# B&R Automation Studio project acoposTrak_simple_control
Automation Studio 4.9.2.46; technology packages: mappMotion 5.12.2, mappView 5.12.1

## Configuration Config1

CPU X20CP3687X, AutomationRuntime C4.90, Build 4.1.2, Vc V4.72.2

### Task classes (Cpu.sw)
```
Cyclic#1 (cycle 2000 us, tolerance 0 us):
  tCTRL_m <- Technology.tCTRL_m.prg
DataObjects: McAcpSys
Binaries: FWRules, McAcpSim, arcoal, arsvcreg, TCData, McAcpDrv, McProfGen, arflatprv, udbdef, iomap, Config_1, arconfig, asfw, ashwac, sysconf, Role, ashwd, User, Config_3, Config_2
Libraries: McBase, McAxis, McAcpTrak, AsBrStr, runtime, astime, fileio, powerlnk, asieccon, standard, asstring
```

### Hardware
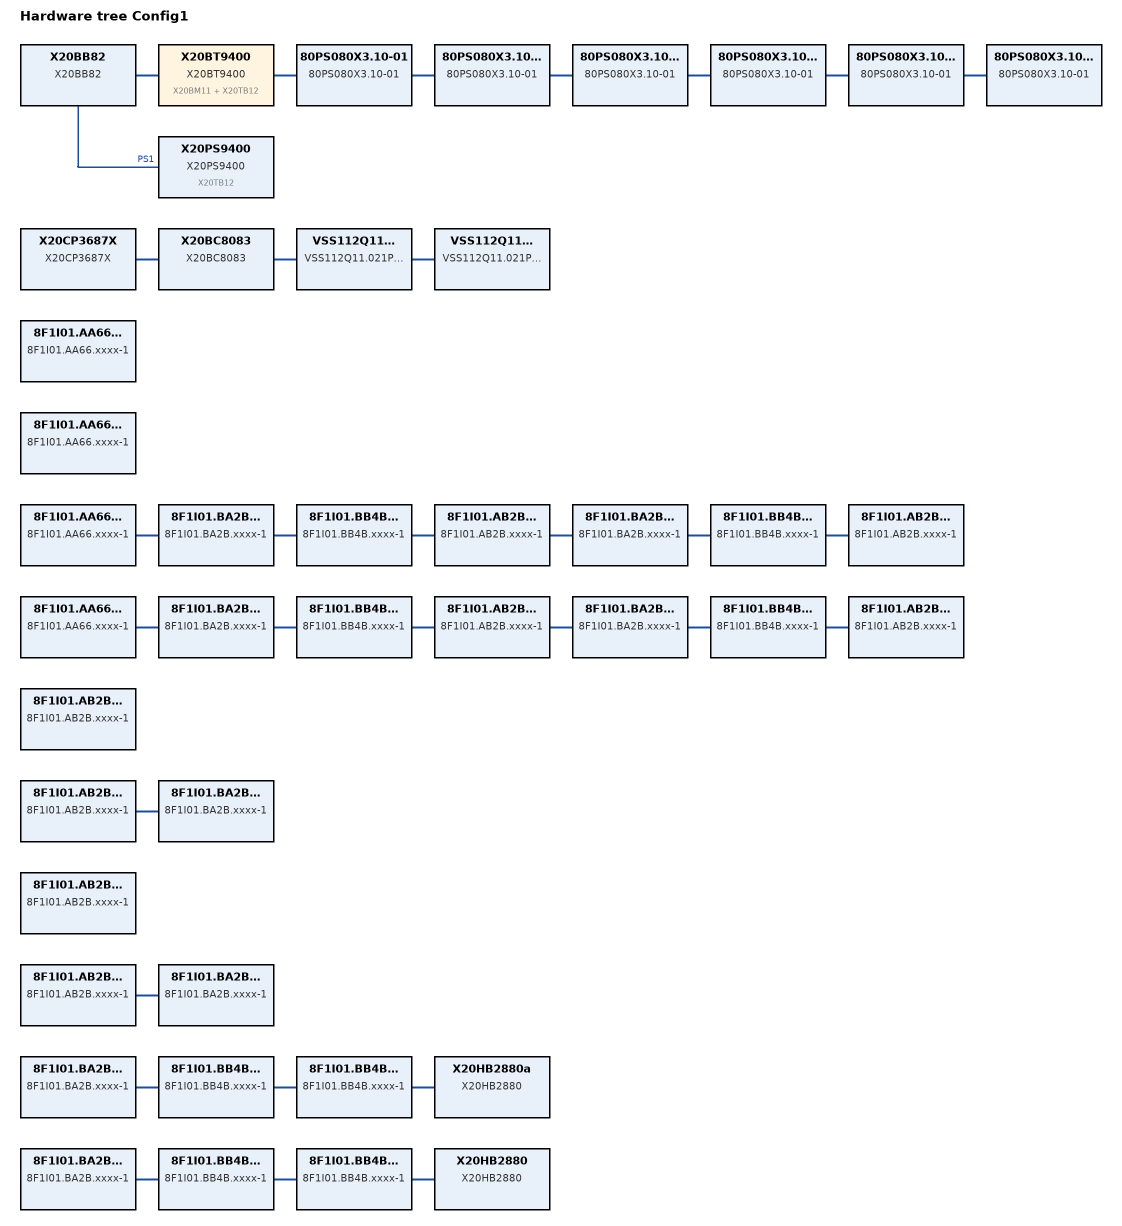
```
80PS080X3.10-01 : 80PS080X3.10-01 v1.3.0.0  [X2X1 -> X20BT9400.X2X1 [Cable Type=X2XCable, Length=10, Version=1.0.0.3]]
  Supervision = off
  VoltageSet01 = 60
80PS080X3.10-01a : 80PS080X3.10-01 v1.3.0.0  [X2X1 -> 80PS080X3.10-01.X2X2 [Cable Type=X2XCable, Length=10, Version=1.0.0.3]]
  ParallelMode01 = on
  VoltageSet01 = 60
80PS080X3.10-01b : 80PS080X3.10-01 v1.3.0.0  [X2X1 -> 80PS080X3.10-01a.X2X2 [Cable Type=X2XCable, Length=10, Version=1.0.0.3]]
  ParallelMode01 = on
  VoltageSet01 = 60
80PS080X3.10-01c : 80PS080X3.10-01 v1.3.0.0  [X2X1 -> 80PS080X3.10-01b.X2X2 [Cable Type=X2XCable, Length=10, Version=1.0.0.3]]
  ParallelMode01 = on
  VoltageSet01 = 60
80PS080X3.10-01d : 80PS080X3.10-01 v1.3.0.0  [X2X1 -> 80PS080X3.10-01c.X2X2 [Cable Type=X2XCable, Length=10, Version=1.0.0.3]]
  ParallelMode01 = on
  VoltageSet01 = 60
80PS080X3.10-01e : 80PS080X3.10-01 v1.3.0.0  [X2X1 -> 80PS080X3.10-01d.X2X2 [Cable Type=X2XCable, Length=10, Version=1.0.0.3]]
  ParallelMode01 = on
  VoltageSet01 = 60
8F1I01.AA66.xxxx-1 : 8F1I01.AA66.xxxx-1 v1.0.0.2  [PLK1 -> 8F1I01.AB2B.xxxx-1.PLK2 [Cable Type=PowerlinkCable, Length=10, Version=1.0.0.3]]
  DriveConfiguration:
    McTypeID = LLMConfig
  DriveConfiguration/Segment:
    Shape = STRAIGHT660
    SegmentReference = Seg_A_1
    StopReaction = UseAssemblySetting
    SpeedFilter = UseAssemblySetting
8F1I01.AA66.xxxx-1a : 8F1I01.AA66.xxxx-1 v1.0.0.2  [PLK1 -> 8F1I01.AB2B.xxxx-1b.PLK2 [Cable Type=PowerlinkCable, Length=10, Version=1.0.0.3]]
  DriveConfiguration:
    McTypeID = LLMConfig
  DriveConfiguration/Segment:
    Shape = STRAIGHT660
    SegmentReference = Seg_A_8
    StopReaction = UseAssemblySetting
    SpeedFilter = UseAssemblySetting
8F1I01.AA66.xxxx-1b : 8F1I01.AA66.xxxx-1 v1.0.0.2  [PLK2 -> 8F1I01.BA2B.xxxx-1g.PLK1 [Cable Type=PowerlinkCable, Length=10, Version=1.0.0.3]]
  DriveConfiguration:
    McTypeID = LLMConfig
  DriveConfiguration/Segment:
    Shape = STRAIGHT660
    SegmentReference = Seg_B_28
    StopReaction = UseAssemblySetting
    SpeedFilter = UseAssemblySetting
8F1I01.AA66.xxxx-1c : 8F1I01.AA66.xxxx-1 v1.0.0.2  [PLK2 -> 8F1I01.BA2B.xxxx-1e.PLK1 (NodeNumber=23) [Cable Type=PowerlinkCable, Length=10, Version=1.0.0.3]]
  DriveConfiguration:
    McTypeID = LLMConfig
  DriveConfiguration/Segment:
    Shape = STRAIGHT660
    SegmentReference = Seg_B_21
    StopReaction = UseAssemblySetting
    SpeedFilter = UseAssemblySetting
8F1I01.AB2B.xxxx-1 : 8F1I01.AB2B.xxxx-1 v1.0.0.2  [PLK1 -> 8F1I01.BA2B.xxxx-1.PLK2 [Cable Type=PowerlinkCable, Length=10, Version=1.0.0.3]; PLK2 -> 8F1I01.AA66.xxxx-1.PLK1 [Cable Type=PowerlinkCable, Length=10, Version=1.0.0.3]]
  DriveConfiguration:
    McTypeID = LLMConfig
  DriveConfiguration/Segment:
    Shape = STRAIGHT105_TO_CIRCULAR
    SegmentReference = Seg_A_2
    StopReaction = UseAssemblySetting
    SpeedFilter = UseAssemblySetting
8F1I01.AB2B.xxxx-1a : 8F1I01.AB2B.xxxx-1 v1.0.0.2  [PLK1 -> 8F1I01.BB4B.xxxx-1.PLK2 (NodeNumber=4) [Cable Type=PowerlinkCable, Length=10, Version=1.0.0.3]; PLK2 -> 8F1I01.BA2B.xxxx-1.PLK1 (NodeNumber=4) [Cable Type=PowerlinkCable, Length=10, Version=1.0.0.3]]
  DriveConfiguration:
    McTypeID = LLMConfig
  DriveConfiguration/Segment:
    Shape = STRAIGHT105_TO_CIRCULAR
    SegmentReference = Seg_A_4
    StopReaction = UseAssemblySetting
    SpeedFilter = UseAssemblySetting
8F1I01.AB2B.xxxx-1b : 8F1I01.AB2B.xxxx-1 v1.0.0.2  [PLK1 -> 8F1I01.BA2B.xxxx-1b.PLK2 [Cable Type=PowerlinkCable, Length=10, Version=1.0.0.3]; PLK2 -> 8F1I01.AA66.xxxx-1a.PLK1 [Cable Type=PowerlinkCable, Length=10, Version=1.0.0.3]]
  DriveConfiguration:
    McTypeID = LLMConfig
  DriveConfiguration/Segment:
    Shape = STRAIGHT105_TO_CIRCULAR
    SegmentReference = Seg_A_9
    StopReaction = UseAssemblySetting
    SpeedFilter = UseAssemblySetting
8F1I01.AB2B.xxxx-1c : 8F1I01.AB2B.xxxx-1 v1.0.0.2  [PLK1 -> 8F1I01.BB4B.xxxx-1b.PLK2 (NodeNumber=10) [Cable Type=PowerlinkCable, Length=10, Version=1.0.0.3]; PLK2 -> 8F1I01.BA2B.xxxx-1b.PLK1 (NodeNumber=10) [Cable Type=PowerlinkCable, Length=10, Version=1.0.0.3]]
  DriveConfiguration:
    McTypeID = LLMConfig
  DriveConfiguration/Segment:
    Shape = STRAIGHT105_TO_CIRCULAR
    SegmentReference = Seg_A_11
    StopReaction = UseAssemblySetting
    SpeedFilter = UseAssemblySetting
8F1I01.AB2B.xxxx-1d : 8F1I01.AB2B.xxxx-1 v1.0.0.2  [PLK1 -> 8F1I01.BB4B.xxxx-1d.PLK2 [Cable Type=PowerlinkCable, Length=10, Version=1.0.0.3]]
  DriveConfiguration:
    McTypeID = LLMConfig
  DriveConfiguration/Segment:
    Shape = STRAIGHT105_TO_CIRCULAR
    SegmentReference = Seg_B_15
    StopReaction = UseAssemblySetting
    SpeedFilter = UseAssemblySetting
8F1I01.AB2B.xxxx-1e : 8F1I01.AB2B.xxxx-1 v1.0.0.2  [PLK1 -> 8F1I01.BB4B.xxxx-1e.PLK2 (NodeNumber=18) [Cable Type=PowerlinkCable, Length=10, Version=1.0.0.3]; PLK2 -> 8F1I01.BA2B.xxxx-1d.PLK1 (NodeNumber=18) [Cable Type=PowerlinkCable, Length=10, Version=1.0.0.3]]
  DriveConfiguration:
    McTypeID = LLMConfig
  DriveConfiguration/Segment:
    Shape = STRAIGHT105_TO_CIRCULAR
    SegmentReference = Seg_B_18
    StopReaction = UseAssemblySetting
    SpeedFilter = UseAssemblySetting
8F1I01.AB2B.xxxx-1f : 8F1I01.AB2B.xxxx-1 v1.0.0.2  [PLK1 -> 8F1I01.BB4B.xxxx-1f.PLK2 (NodeNumber=29) [Cable Type=PowerlinkCable, Length=10, Version=1.0.0.3]]
  DriveConfiguration:
    McTypeID = LLMConfig
  DriveConfiguration/Segment:
    Shape = STRAIGHT105_TO_CIRCULAR
    SegmentReference = Seg_B_22
    StopReaction = UseAssemblySetting
    SpeedFilter = UseAssemblySetting
8F1I01.AB2B.xxxx-1g : 8F1I01.AB2B.xxxx-1 v1.0.0.2  [PLK1 -> 8F1I01.BB4B.xxxx-1g.PLK2 [Cable Type=PowerlinkCable, Length=10, Version=1.0.0.3]; PLK2 -> 8F1I01.BA2B.xxxx-1f.PLK1 [Cable Type=PowerlinkCable, Length=10, Version=1.0.0.3]]
  DriveConfiguration:
    McTypeID = LLMConfig
  DriveConfiguration/Segment:
    Shape = STRAIGHT105_TO_CIRCULAR
    SegmentReference = Seg_B_25
    StopReaction = UseAssemblySetting
    SpeedFilter = UseAssemblySetting
8F1I01.BA2B.xxxx-1 : 8F1I01.BA2B.xxxx-1 v1.0.0.2  [PLK1 -> 8F1I01.AB2B.xxxx-1a.PLK2 [Cable Type=PowerlinkCable, Length=10, Version=1.0.0.3]; PLK2 -> 8F1I01.AB2B.xxxx-1.PLK1 [Cable Type=PowerlinkCable, Length=10, Version=1.0.0.3]]
  DriveConfiguration:
    McTypeID = LLMConfig
  DriveConfiguration/Segment:
    Shape = CIRCULAR_TO_STRAIGHT105
    SegmentReference = Seg_A_3
    StopReaction = UseAssemblySetting
    SpeedFilter = UseAssemblySetting
8F1I01.BA2B.xxxx-1a : 8F1I01.BA2B.xxxx-1 v1.0.0.2  [PLK2 -> 8F1I01.BB4B.xxxx-1a.PLK1 (NodeNumber=9) [Cable Type=PowerlinkCable, Length=10, Version=1.0.0.3]]
  DriveConfiguration:
    McTypeID = LLMConfig
  DriveConfiguration/Segment:
    Shape = CIRCULAR_TO_STRAIGHT105
    SegmentReference = Seg_A_7
    StopReaction = UseAssemblySetting
    SpeedFilter = UseAssemblySetting
8F1I01.BA2B.xxxx-1b : 8F1I01.BA2B.xxxx-1 v1.0.0.2  [PLK1 -> 8F1I01.AB2B.xxxx-1c.PLK2 [Cable Type=PowerlinkCable, Length=10, Version=1.0.0.3]; PLK2 -> 8F1I01.AB2B.xxxx-1b.PLK1 [Cable Type=PowerlinkCable, Length=10, Version=1.0.0.3]]
  DriveConfiguration:
    McTypeID = LLMConfig
  DriveConfiguration/Segment:
    Shape = CIRCULAR_TO_STRAIGHT105
    SegmentReference = Seg_A_10
    StopReaction = UseAssemblySetting
    SpeedFilter = UseAssemblySetting
8F1I01.BA2B.xxxx-1c : 8F1I01.BA2B.xxxx-1 v1.0.0.2  [PLK2 -> 8F1I01.BB4B.xxxx-1c.PLK1 (NodeNumber=15) [Cable Type=PowerlinkCable, Length=10, Version=1.0.0.3]]
  DriveConfiguration:
    McTypeID = LLMConfig
  DriveConfiguration/Segment:
    Shape = CIRCULAR_TO_STRAIGHT105
    SegmentReference = Seg_A_14
    StopReaction = UseAssemblySetting
    SpeedFilter = UseAssemblySetting
8F1I01.BA2B.xxxx-1d : 8F1I01.BA2B.xxxx-1 v1.0.0.2  [PLK1 -> 8F1I01.AB2B.xxxx-1e.PLK2 [Cable Type=PowerlinkCable, Length=10, Version=1.0.0.3]; PLK2 -> 8F1I01.BB4B.xxxx-1d.PLK1 [Cable Type=PowerlinkCable, Length=10, Version=1.0.0.3]]
  DriveConfiguration:
    McTypeID = LLMConfig
  DriveConfiguration/Segment:
    Shape = CIRCULAR_TO_STRAIGHT105
    SegmentReference = Seg_B_17
    StopReaction = UseAssemblySetting
    SpeedFilter = UseAssemblySetting
8F1I01.BA2B.xxxx-1e : 8F1I01.BA2B.xxxx-1 v1.0.0.2  [PLK1 -> 8F1I01.AA66.xxxx-1c.PLK2 (NodeNumber=22) [Cable Type=PowerlinkCable, Length=10, Version=1.0.0.3]; PLK2 -> 8F1I01.BB4B.xxxx-1e.PLK1 (NodeNumber=22) [Cable Type=PowerlinkCable, Length=10, Version=1.0.0.3]]
  DriveConfiguration:
    McTypeID = LLMConfig
  DriveConfiguration/Segment:
    Shape = CIRCULAR_TO_STRAIGHT105
    SegmentReference = Seg_B_20
    StopReaction = UseAssemblySetting
    SpeedFilter = UseAssemblySetting
8F1I01.BA2B.xxxx-1f : 8F1I01.BA2B.xxxx-1 v1.0.0.2  [PLK1 -> 8F1I01.AB2B.xxxx-1g.PLK2 (NodeNumber=24) [Cable Type=PowerlinkCable, Length=10, Version=1.0.0.3]; PLK2 -> 8F1I01.BB4B.xxxx-1f.PLK1 (NodeNumber=24) [Cable Type=PowerlinkCable, Length=10, Version=1.0.0.3]]
  DriveConfiguration:
    McTypeID = LLMConfig
  DriveConfiguration/Segment:
    Shape = CIRCULAR_TO_STRAIGHT105
    SegmentReference = Seg_B_24
    StopReaction = UseAssemblySetting
    SpeedFilter = UseAssemblySetting
8F1I01.BA2B.xxxx-1g : 8F1I01.BA2B.xxxx-1 v1.0.0.2  [PLK1 -> 8F1I01.AA66.xxxx-1b.PLK2 [Cable Type=PowerlinkCable, Length=10, Version=1.0.0.3]; PLK2 -> 8F1I01.BB4B.xxxx-1g.PLK1 [Cable Type=PowerlinkCable, Length=10, Version=1.0.0.3]]
  DriveConfiguration:
    McTypeID = LLMConfig
  DriveConfiguration/Segment:
    Shape = CIRCULAR_TO_STRAIGHT105
    SegmentReference = Seg_B_27
    StopReaction = UseAssemblySetting
    SpeedFilter = UseAssemblySetting
8F1I01.BB4B.xxxx-1 : 8F1I01.BB4B.xxxx-1 v1.0.0.2  [PLK1 -> 8F1I01.BB4B.xxxx-1a.PLK2 (NodeNumber=3) [Cable Type=PowerlinkCable, Length=10, Version=1.0.0.3]; PLK2 -> 8F1I01.AB2B.xxxx-1a.PLK1 (NodeNumber=3) [Cable Type=PowerlinkCable, Length=10, Version=1.0.0.3]; PLK3 -> X20HB2880a.ETH1 (NodeNumber=3) [Cable Type=PowerlinkCable, Length=10, Version=1.0.0.3]]
  EPL_Chained = on
  EnableDNA = on
  DriveConfiguration:
    McTypeID = LLMConfig
  DriveConfiguration/Segment:
    Shape = CIRCULAR
    SegmentReference = Seg_A_5
    StopReaction = UseAssemblySetting
    SpeedFilter = UseAssemblySetting
8F1I01.BB4B.xxxx-1a : 8F1I01.BB4B.xxxx-1 v1.0.0.2  [PLK1 -> 8F1I01.BA2B.xxxx-1a.PLK2 (NodeNumber=8) [Cable Type=PowerlinkCable, Length=10, Version=1.0.0.3]; PLK2 -> 8F1I01.BB4B.xxxx-1.PLK1 (NodeNumber=8) [Cable Type=PowerlinkCable, Length=10, Version=1.0.0.3]]
  DriveConfiguration:
    McTypeID = LLMConfig
  DriveConfiguration/Segment:
    Shape = CIRCULAR
    SegmentReference = Seg_A_6
    StopReaction = UseAssemblySetting
    SpeedFilter = UseAssemblySetting
8F1I01.BB4B.xxxx-1b : 8F1I01.BB4B.xxxx-1 v1.0.0.2  [PLK1 -> 8F1I01.BB4B.xxxx-1c.PLK2 (NodeNumber=2) [Cable Type=PowerlinkCable, Length=10, Version=1.0.0.3]; PLK2 -> 8F1I01.AB2B.xxxx-1c.PLK1 (NodeNumber=2) [Cable Type=PowerlinkCable, Length=10, Version=1.0.0.3]; PLK3 -> X20HB2880.ETH1 (NodeNumber=2) [Cable Type=PowerlinkCable, Length=10, Version=1.0.0.3]]
  EPL_Chained = on
  EnableDNA = on
  DriveConfiguration:
    McTypeID = LLMConfig
  DriveConfiguration/Segment:
    Shape = CIRCULAR
    SegmentReference = Seg_A_12
    StopReaction = UseAssemblySetting
    SpeedFilter = UseAssemblySetting
8F1I01.BB4B.xxxx-1c : 8F1I01.BB4B.xxxx-1 v1.0.0.2  [PLK1 -> 8F1I01.BA2B.xxxx-1c.PLK2 (NodeNumber=14) [Cable Type=PowerlinkCable, Length=10, Version=1.0.0.3]; PLK2 -> 8F1I01.BB4B.xxxx-1b.PLK1 (NodeNumber=14) [Cable Type=PowerlinkCable, Length=10, Version=1.0.0.3]]
  DriveConfiguration:
    McTypeID = LLMConfig
  DriveConfiguration/Segment:
    Shape = CIRCULAR
    SegmentReference = Seg_A_13
    StopReaction = UseAssemblySetting
    SpeedFilter = UseAssemblySetting
8F1I01.BB4B.xxxx-1d : 8F1I01.BB4B.xxxx-1 v1.0.0.2  [PLK1 -> 8F1I01.BA2B.xxxx-1d.PLK2 [Cable Type=PowerlinkCable, Length=10, Version=1.0.0.3]; PLK2 -> 8F1I01.AB2B.xxxx-1d.PLK1 [Cable Type=PowerlinkCable, Length=10, Version=1.0.0.3]]
  DriveConfiguration:
    McTypeID = LLMConfig
  DriveConfiguration/Segment:
    Shape = CIRCULAR
    SegmentReference = Seg_B_16
    StopReaction = UseAssemblySetting
    SpeedFilter = UseAssemblySetting
8F1I01.BB4B.xxxx-1e : 8F1I01.BB4B.xxxx-1 v1.0.0.2  [PLK1 -> 8F1I01.BA2B.xxxx-1e.PLK2 (NodeNumber=17) [Cable Type=PowerlinkCable, Length=10, Version=1.0.0.3]; PLK2 -> 8F1I01.AB2B.xxxx-1e.PLK1 (NodeNumber=17) [Cable Type=PowerlinkCable, Length=10, Version=1.0.0.3]; PLK3 -> X20HB2880.ETH2 (NodeNumber=17) [Cable Type=PowerlinkCable, Length=10, Version=1.0.0.3]]
  EPL_Chained = on
  EnableDNA = on
  DriveConfiguration:
    McTypeID = LLMConfig
  DriveConfiguration/Segment:
    Shape = CIRCULAR
    SegmentReference = Seg_B_19
    StopReaction = UseAssemblySetting
    SpeedFilter = UseAssemblySetting
8F1I01.BB4B.xxxx-1f : 8F1I01.BB4B.xxxx-1 v1.0.0.2  [PLK1 -> 8F1I01.BA2B.xxxx-1f.PLK2 (NodeNumber=16) [Cable Type=PowerlinkCable, Length=10, Version=1.0.0.3]; PLK2 -> 8F1I01.AB2B.xxxx-1f.PLK1 (NodeNumber=16) [Cable Type=PowerlinkCable, Length=10, Version=1.0.0.3]; PLK3 -> X20HB2880a.ETH2 (NodeNumber=16) [Cable Type=PowerlinkCable, Length=10, Version=1.0.0.3]]
  EPL_Chained = on
  EnableDNA = on
  DriveConfiguration:
    McTypeID = LLMConfig
  DriveConfiguration/Segment:
    Shape = CIRCULAR
    SegmentReference = Seg_B_23
    StopReaction = UseAssemblySetting
    SpeedFilter = UseAssemblySetting
8F1I01.BB4B.xxxx-1g : 8F1I01.BB4B.xxxx-1 v1.0.0.2  [PLK1 -> 8F1I01.BA2B.xxxx-1g.PLK2 [Cable Type=PowerlinkCable, Length=10, Version=1.0.0.3]; PLK2 -> 8F1I01.AB2B.xxxx-1g.PLK1 [Cable Type=PowerlinkCable, Length=10, Version=1.0.0.3]]
  DriveConfiguration:
    McTypeID = LLMConfig
  DriveConfiguration/Segment:
    Shape = CIRCULAR
    SegmentReference = Seg_B_26
    StopReaction = UseAssemblySetting
    SpeedFilter = UseAssemblySetting
VSS112Q11.021P-000 : VSS112Q11.021P-000 v1.1.0.284  [PLK1 -> X20BC8083.PLK2 (NodeNumber=30) [Cable Type=PowerlinkCable, Length=10, Version=1.0.0.3]; PLK2 -> VSS112Q11.021P-000a.PLK1 (NodeNumber=30) [Cable Type=PowerlinkCable, Length=10, Version=1.0.0.3]]
VSS112Q11.021P-000a : VSS112Q11.021P-000 v1.1.0.284  [PLK1 -> VSS112Q11.021P-000.PLK2 (NodeNumber=31) [Cable Type=PowerlinkCable, Length=10, Version=1.0.0.3]]
X20BB82 : X20BB82 v1.0.3.0
X20BC8083 : X20BC8083 v2.11.1.0  [PLK1 -> X20CP3687X.IF3 (NodeNumber=1) [Cable Type=PowerlinkCable, Length=10, Version=1.0.0.3]; PLK2 -> VSS112Q11.021P-000.PLK1 (NodeNumber=1) [Cable Type=PowerlinkCable, Length=10, Version=1.0.0.3]; SL -> X20BB82.SL1]
  EnableDNA = on
X20BM11 : X20BM11 v1.0.0.1  [X2X1 -> X20BB82.IF1]
X20BT9400 : X20BT9400 v1.1.0.0  [SS1 -> X20TB12a.SS; SL -> X20BM11.SL1]
X20CP3687X : X20CP3687X v1.1.2.0
  Connector IF2:
    ActivateDevice = 1
  ConfigurationID = acoposTrak_simple_control_Config1
  Simulation = 1
  SystemTick = 2000
  TaskClassIdleTime = 2000
  Cyclic1Duration = 2000
  Cyclic1Tolerance = 0
  FileDevice1
  FileDeviceName1 = SvgData
  FileDevicePath1 = C:\Users\romanp\Downloads\Trak\
  FileDevice2
  FileDeviceName2 = User
  FileDevicePath2 = C:\Users\romanp\Downloads\Trak\
  ActivateOpcUa = 1
  OpcUaInformationModels_PV_Version = 1
X20HB2880 : X20HB2880 v1.1.2.0  [ETH1 -> 8F1I01.BB4B.xxxx-1b.PLK3 [Cable Type=PowerlinkCable, Length=10, Version=1.0.0.3]; ETH2 -> 8F1I01.BB4B.xxxx-1e.PLK3 [Cable Type=PowerlinkCable, Length=10, Version=1.0.0.3]; SS -> X20BB82.SS1]
X20HB2880a : X20HB2880 v1.1.2.0  [ETH1 -> 8F1I01.BB4B.xxxx-1.PLK3 [Cable Type=PowerlinkCable, Length=10, Version=1.0.0.3]; ETH2 -> 8F1I01.BB4B.xxxx-1f.PLK3 [Cable Type=PowerlinkCable, Length=10, Version=1.0.0.3]; SS -> X20BB82.SS2]
X20PS9400 : X20PS9400 v1.4.0.0  [SS1 -> X20TB12.SS; PS -> X20BB82.PS1]
X20TB12 : X20TB12 v1.0.0.0
X20TB12a : X20TB12 v1.0.0.0
```

### Config_1.assembly - X20CP3687X/mappMotion/TrakOval/Config_1.assembly
```
Element gAssembly_1 (Type=assembly)
  Tracks:
    TrackSeparation = 0.030
    Track[1]:
      Segments:
        SegmentRef[1] = ::Seg_A_1
        SegmentRef[2] = ::Seg_A_2
        SegmentRef[3] = ::Seg_A_3
        SegmentRef[4] = ::Seg_A_4
        SegmentRef[5] = ::Seg_A_5
        SegmentRef[6] = ::Seg_A_6
        SegmentRef[7] = ::Seg_A_7
        SegmentRef[8] = ::Seg_A_8
        SegmentRef[9] = ::Seg_A_9
        SegmentRef[10] = ::Seg_A_10
        SegmentRef[11] = ::Seg_A_11
        SegmentRef[12] = ::Seg_A_12
        SegmentRef[13] = ::Seg_A_13
        SegmentRef[14] = ::Seg_A_14
      Position = Absolute
        SegmentRef = 
        SegmentCountDirection = RightToLeft
        Translation:
          X = 0.0
          Y = 0.0
          Z = 0.0
        Orientation:
          Angle1 = 0.0
          Angle2 = 0.0
          Angle3 = 180
    Track[2]:
      Segments:
        SegmentRef[1] = ::Seg_B_15
        SegmentRef[2] = ::Seg_B_16
        SegmentRef[3] = ::Seg_B_17
        SegmentRef[4] = ::Seg_B_18
        SegmentRef[5] = ::Seg_B_19
        SegmentRef[6] = ::Seg_B_20
        SegmentRef[7] = ::Seg_B_21
        SegmentRef[8] = ::Seg_B_22
        SegmentRef[9] = ::Seg_B_23
        SegmentRef[10] = ::Seg_B_24
        SegmentRef[11] = ::Seg_B_25
        SegmentRef[12] = ::Seg_B_26
        SegmentRef[13] = ::Seg_B_27
        SegmentRef[14] = ::Seg_B_28
      Position = RelativeToOne
        TrackSegmentPosition:
          SegmentRef = ::Seg_B_15
        Base:
          SegmentRef = ::Seg_A_1
  CommonSegmentSettings:
    SegmentSimulationOnPLC = Off
    StopReaction = InductionHalt
    SpeedFilter = NotUsed
    ControllerParameters:
      DefaultParameter:
        Controller:
          Position:
            ProportionalGain = 200
          Speed:
            ProportionalGain = 80
            IntegrationTime = 0.0
          FeedForward:
            TotalMass = 1
            ForcePositive = 0.0
            ForceNegative = 0.0
            SpeedForceFactor = 0.0
            ForceLoad = 0.0
        MovementErrorLimits:
          PositionError = 0.001
          VelocityError = 0.05
      AdditionalParameterSets = NotUsed
    ShuttleIdentificationTime = 0
  Shuttles:
    MaxShuttleCount = 10
    DistanceReserve:
      Collision = 0.002
      ErrorStop = 0.006
    ShuttleStereotypes:
      ShuttleStRef[1] = ShuttleStereotype_1
    MagnetPlateConfigurations:
      ShuttleType[1] = 8F1SA.100.xxxxxx-x
    CollisionAvoidance:
      Strategy = Constant
      MaximumModelDimensions:
        Length:
          ExtentToFront = 0.04
          ExtentToBack = 0.04
        Width:
          Width = 0.040
  Visualization:
    MonitoringPv = ::gShuttleMon
    ProcessingTaskClass = 1
```

### Config_2.shuttlestereotype - X20CP3687X/mappMotion/TrakOval/Config_2.shuttlestereotype
```
Element ShuttleStereotype_1 (Type=shuttlestereotype)
  MeasurementUnit = 5067858
  MeasurementResolution = 0.00001
  MovementLimits = Internal
    VelocityIsReadOnly = 0
    Velocity:
      Velocity = 4
    AccelerationIsReadOnly = 0
    Acceleration:
      Acceleration = 40
    DecelerationIsReadOnly = 0
    Deceleration:
      Deceleration = 40
  JerkFilter = NotUsed
  UserData:
    Size = 12
```

### Config_3.sector - X20CP3687X/mappMotion/TrakOval/Config_3.sector
```
Element SectorTrackA (Type=sector)
  Type = Composed
    StartSegment:
      SegmentRef = ::Seg_A_1
    IntermediateSegments:
      SegmentRef[1] = ::Seg_A_2
      SegmentRef[2] = ::Seg_A_3
      SegmentRef[3] = ::Seg_A_4
      SegmentRef[4] = ::Seg_A_5
      SegmentRef[5] = ::Seg_A_6
      SegmentRef[6] = ::Seg_A_7
      SegmentRef[7] = ::Seg_A_8
      SegmentRef[8] = ::Seg_A_9
      SegmentRef[9] = ::Seg_A_10
      SegmentRef[10] = ::Seg_A_11
      SegmentRef[11] = ::Seg_A_12
      SegmentRef[12] = ::Seg_A_13
    EndSegment:
      SegmentRef = ::Seg_A_14
      PositionRelativeTo = FromEnd
Element SectorTrackB (Type=sector)
  Type = Composed
    StartSegment:
      SegmentRef = ::Seg_B_28
    IntermediateSegments:
      SegmentRef[1] = ::Seg_B_15
      SegmentRef[2] = ::Seg_B_16
      SegmentRef[3] = ::Seg_B_17
      SegmentRef[4] = ::Seg_B_18
      SegmentRef[5] = ::Seg_B_19
      SegmentRef[6] = ::Seg_B_20
      SegmentRef[7] = ::Seg_B_21
      SegmentRef[8] = ::Seg_B_22
      SegmentRef[9] = ::Seg_B_23
      SegmentRef[10] = ::Seg_B_24
      SegmentRef[11] = ::Seg_B_25
      SegmentRef[12] = ::Seg_B_26
    EndSegment:
      SegmentRef = ::Seg_B_27
      PositionRelativeTo = FromEnd
```

## Logical view

Binary libraries used (declarations not repeated): operator, runtime, astime, AsIecCon, McBase 5.12.2, McAxis 5.12.2, McAcpTrak 5.12.2, AsBrStr, standard, asstring

### Global.var - Global variables
```iecst
VAR
	gShuttleMon : McAcpTrakAssemblyMonData;
	Seg_A_1 : McSegmentType;
	Seg_A_2 : McSegmentType;
	Seg_A_3 : McSegmentType;
	Seg_A_4 : McSegmentType;
	Seg_A_5 : McSegmentType;
	Seg_A_6 : McSegmentType;
	Seg_A_7 : McSegmentType;
	Seg_A_8 : McSegmentType;
	Seg_A_9 : McSegmentType;
	Seg_A_10 : McSegmentType;
	Seg_A_11 : McSegmentType;
	Seg_A_12 : McSegmentType;
	Seg_A_13 : McSegmentType;
	Seg_A_14 : McSegmentType;
	Seg_B_15 : McSegmentType;
	Seg_B_16 : McSegmentType;
	Seg_B_17 : McSegmentType;
	Seg_B_18 : McSegmentType;
	Seg_B_19 : McSegmentType;
	Seg_B_20 : McSegmentType;
	Seg_B_21 : McSegmentType;
	Seg_B_22 : McSegmentType;
	Seg_B_23 : McSegmentType;
	Seg_B_24 : McSegmentType;
	Seg_B_25 : McSegmentType;
	Seg_B_26 : McSegmentType;
	Seg_B_27 : McSegmentType;
	Seg_B_28 : McSegmentType;
END_VAR
```


### Program Logical/Technology/tCTRL_m (ANSIC)

#### Main.c - Init, cyclic, exit code
```c
/**
 * MIT License
 * Copyright(c) 2021 Roman Parak
 * Permission is hereby granted, free of charge, to any person obtaining a copy
 * of this software and associated documentation files (the "Software"), to deal
 * in the Software without restriction, including without limitation the rights
 * to use, copy, modify, merge, publish, distribute, sublicense, and/or sell
 * copies of the Software, and to permit persons to whom the Software is
 * furnished to do so, subject to the following conditions:
 * The above copyright notice and this permission notice shall be included in all
 * copies or substantial portions of the Software.
 * THE SOFTWARE IS PROVIDED "AS IS", WITHOUT WARRANTY OF ANY KIND, EXPRESS OR
 * IMPLIED, INCLUDING BUT NOT LIMITED TO THE WARRANTIES OF MERCHANTABILITY,
 * FITNESS FOR A PARTICULAR PURPOSE AND NONINFRINGEMENT. IN NO EVENT SHALL THE
 * AUTHORS OR COPYRIGHT HOLDERS BE LIABLE FOR ANY CLAIM, DAMAGES OR OTHER
 * LIABILITY, WHETHER IN AN ACTION OF CONTRACT, TORT OR OTHERWISE, ARISING FROM,
 * OUT OF OR IN CONNECTION WITH THE SOFTWARE OR THE USE OR OTHER DEALINGS IN THE
 * SOFTWARE.
 */

/**
 * Author   : Roman Parak
 * Email    : Roman.Parak@outlook.com
 * File Name: Main.c
 * Github   : https://github.com/rparak
 */

/** < Include B&R Automation libraries (declarations for B&R ANSI C extensions) */
#include <bur/plctypes.h>

#ifdef _DEFAULT_INCLUDES
#include <AsDefault.h>
#endif

/** < Include header file with specified structures / enums, etc. */
#include "Main.h"

/**
 * Declaration of auxiliary functions
 * See the header file for more information -> 'Main.h'
 */

/// Reset parameters, environment, etc.
void reset_shuttle_param(USINT num_of_shuttles, USINT initial_sector, REAL offset);
void reset_env();
/// Cyclic reading shuttle parameters (position, velocity, etc.)
void read_shuttle_param(USINT num_of_shuttles, REAL offset);
/// Axis motion control functions (parameters, mode, etc.)
void set_animation_mode();
void set_shuttle_move_param(USINT index, USINT sector, LREAL position, REAL velocity);
/// Auxiliary functions for calculating the maximum/minimum position index of the shuttle.
USINT min_number_index(USINT num_of_shuttles, LREAL machine_vision_position, USINT sector);
USINT max_number_index(USINT num_of_shuttles, LREAL machine_vision_position, USINT sector);

/**
 * Program Intitialization
 */
void _INIT ProgramInit(void)
{
	/// Initialization of function block inputs
	MC_BR_AsmPowerOn_AcpTrak_0.Assembly       = &gAssembly_1;
	MC_BR_AsmGetShuttle_AcpTrak_0.Assembly    = &gAssembly_1;
	MC_BR_AsmPowerOff_AcpTrak_0.Assembly      = &gAssembly_1;
	MC_BR_AsmReadStatus_AcpTrak_0.Enable = 1;
	MC_BR_AsmReadStatus_AcpTrak_0.Assembly    = &gAssembly_1;
	MC_BR_AsmReset_AcpTrak_0.Assembly         = &gAssembly_1;
	MC_BR_AsmDeleteShuttle_AcpTrak_0.Assembly = &gAssembly_1;

	/// Set initialization parameters of the structure for custom structure (ACOPOStrak control and data collection).
	gTrakAsm.shuttle.num_of_shuttles  = 6;
	gTrakAsm.shuttle.shuttle_offset   = 0.2;
	gTrakAsm.shuttle.shuttle_velocity = 1.5;
	gTrakAsm.shuttle.sector_legth     = 5.885136451852274;
	gTrakAsm.actual_state             = ACPt_CTRL_POWER_OFF;

	/// Set machine vision camera (digital-twin) position (0 - Sector A, 1 - Sector B)
	dt_service.machine_vision_position[0] = 4.45;
	dt_service.machine_vision_position[1] = 4.75;
}

/**
 * Program Cyclic
 *
 * Duration (Cycle Time): 2000 [µs]
 * Tolerance            : 0    [µs]
 */
void _CYCLIC ProgramCyclic(void)
{
	/**
	 * Main state machine for control of a ACOPOStrak.
	 *
	 * Number of states: 15 (for more information -> 'Main.h')
	 * Structure: acoposT_ctrl_state_enum
	 */

	switch(gTrakAsm.actual_state){
		case ACPt_CTRL_POWER_OFF: ///< Turn off the axes and reset each of the parameters.
			{
				/// reset some status parameters
				gTrakAsm.status.power_on 	   = 0;
				gTrakAsm.status.is_homed       = 0;
				gTrakAsm.status.shuttles_exist = 0;
				/// enable the user to select initial parameters
				mv_service.enable_param 	   = 1;

				/// reset other parameters (for more information -> 'Main.h')
				reset_shuttle_param(gTrakAsm.shuttle.num_of_shuttles, gTrakAsm.shuttle.initial_sector, gTrakAsm.shuttle.shuttle_offset);
				reset_env();

				if(MC_BR_AsmPowerOff_AcpTrak_0.Done == 1){
					MC_BR_AsmPowerOff_AcpTrak_0.Execute = 0;
				}else if(gTrakAsm.control.power == 1){
					mv_service.enable_param = 0;
					gTrakAsm.actual_state = ACPt_CTRL_POWER_ON;
				}
			}
			break;

		case ACPt_CTRL_POWER_ON: ///< Turn on each of the axes.
			{
				MC_BR_AsmPowerOn_AcpTrak_0.Execute = 1;

				if(MC_BR_AsmPowerOn_AcpTrak_0.Done == 1){
					gTrakAsm.status.power_on      = 1;
					gTrakAsm.status.shuttle_index = 0;
					gTrakAsm.actual_state = ACPt_CTRL_ADD_SHUTTLE_1;
				}
			}
			break;

		case ACPt_CTRL_ADD_SHUTTLE_1: ///< Adding Shuttle for simulation.
			{
				if(gTrakAsm.status.shuttle_index < gTrakAsm.shuttle.num_of_shuttles){
					if(gTrakAsm.shuttle.parameter[gTrakAsm.status.shuttle_index].sector_number == 0){
						MC_BR_SecAddShuttle_AcpTrak_0.Sector   = &SectorTrackA;
					}else if(gTrakAsm.shuttle.parameter[gTrakAsm.status.shuttle_index].sector_number == 1){
						MC_BR_SecAddShuttle_AcpTrak_0.Sector   = &SectorTrackB;
					}

					MC_BR_SecAddShuttle_AcpTrak_0.Execute  					  = 1;
					MC_BR_SecAddShuttle_AcpTrak_0.Position 			          = gTrakAsm.shuttle.parameter[gTrakAsm.status.shuttle_index].initial_position;
					MC_BR_SecAddShuttle_AcpTrak_0.AdvancedParameters.Velocity = 0.0;

					gTrakAsm.actual_state = ACPt_CTRL_ADD_SHUTTLE_2;
				}else{
					gTrakAsm.actual_state = ACPt_CTRL_GET_SHUTTLE_1;
				}

			}
			break;

		case ACPt_CTRL_ADD_SHUTTLE_2: ///< When the shuttle is added correctly, increase the index by one.
			{
				if(MC_BR_SecAddShuttle_AcpTrak_0.Done == 1){
					gTrakAsm.status.shuttle_index++;
					gTrakAsm.actual_state = ACPt_CTRL_ADD_SHUTTLE_1;
				}
			}
			break;

		case ACPt_CTRL_GET_SHUTTLE_1: ///< Get all available assembly information. (Initialization State)
			{
				MC_BR_AsmGetShuttle_AcpTrak_0.Enable = 1;
				MC_BR_AsmGetShuttle_AcpTrak_0.Next   = 0;
				gTrakAsm.status.shuttle_index = 0;
				gTrakAsm.actual_state 		  = ACPt_CTRL_GET_SHUTTLE_3;

			}
			break;

		case ACPt_CTRL_GET_SHUTTLE_2: ///< Get all available assembly information. (Get next shuttle information)
			{
				MC_BR_AsmGetShuttle_AcpTrak_0.Next = 1;
				gTrakAsm.actual_state = ACPt_CTRL_GET_SHUTTLE_3;
			}
			break;

		case ACPt_CTRL_GET_SHUTTLE_3: ///< Get all available assembly information. (When the shuttle is exist, increase the index by one)
			{
				if(MC_BR_AsmGetShuttle_AcpTrak_0.Valid == 1){
					gTrakAsm.shuttle_axis[gTrakAsm.status.shuttle_index] = MC_BR_AsmGetShuttle_AcpTrak_0.Axis;
					gTrakAsm.status.shuttle_index++;

					if(MC_BR_AsmGetShuttle_AcpTrak_0.RemainingCount == 0){
						MC_BR_AsmGetShuttle_AcpTrak_0.Enable = 0;
						gTrakAsm.status.shuttles_exist = 1;
						gTrakAsm.actual_state 		   = ACPt_CTRL_WAIT;
					}else{
						MC_BR_AsmGetShuttle_AcpTrak_0.Next = 0;
						gTrakAsm.actual_state = ACPt_CTRL_GET_SHUTTLE_2;
					}
				}
			}
			break;

		case ACPt_CTRL_WAIT: ///< Wait for command from HMI visualization (user).
			{
				gTrakAsm.status.shuttle_index = 0;
				gTrakAsm.status.is_homed      = 1;

				/// Main state machine for animation mode control of a ACOPOStrak. -> (for more information -> 'Main.h')
				set_animation_mode();
				/// Reading shuttle parameters (position, velocity, etc.) -> (for more information -> 'Main.h')
				read_shuttle_param(gTrakAsm.shuttle.num_of_shuttles, gTrakAsm.shuttle.shuttle_offset);

				/**
				* Read the user commands from the HMI and switch to the appropriate state.
				*
				* *.reset_evn: Delete each of the shuttles and return to the initial state (Power Off)
				* *.shuttle_start: Start moving from user-selected parameters.
				* *.shuttle_stop: Stop moving. The braking distance is initialized in the configuration file (Configuration File / mappMotion / ...)
				*/

				if(gTrakAsm.control.reset_evn == 1){
					gTrakAsm.control.power = 0;
					MC_BR_AsmPowerOff_AcpTrak_0.Execute = 1;
					gTrakAsm.actual_state = ACPt_CTRL_DELETE;
				}else if(gTrakAsm.control.shuttle_start == 1){
					gTrakAsm.control.shuttle_start = 0;
					if(gTrakAsm.shuttle.move_type == 0){
						gTrakAsm.actual_state = ACPt_CTRL_MOVE_VEL_1;
					}else if(gTrakAsm.shuttle.move_type == 1){
						gTrakAsm.actual_state = ACPt_CTRL_MOVE_POS_1;
					}
				}else if(gTrakAsm.control.shuttle_stop == 1){
					gTrakAsm.control.shuttle_stop = 0;
					gTrakAsm.actual_state = ACPt_CTRL_STOPPING;
				}
			}
			break;

		case ACPt_CTRL_MOVE_VEL_1: ///< Velocity control of the axes.
			{

				if(gTrakAsm.status.shuttle_index >= gTrakAsm.shuttle.num_of_shuttles){
					gTrakAsm.actual_state = ACPt_CTRL_WAIT;
				}else if(gTrakAsm.shuttle_axis[gTrakAsm.status.shuttle_index].controlif != 0){
					MC_BR_RoutedMoveVel_AcpTrak_0.Axis    = &gTrakAsm.shuttle_axis[gTrakAsm.status.shuttle_index];
					MC_BR_RoutedMoveVel_AcpTrak_0.Execute = 1;

					if(gTrakAsm.shuttle.parameter[gTrakAsm.status.shuttle_index].sector_number == 0){
						MC_BR_RoutedMoveVel_AcpTrak_0.Sector = &SectorTrackA;
					}else if(gTrakAsm.shuttle.parameter[gTrakAsm.status.shuttle_index].sector_number == 1){
						MC_BR_RoutedMoveVel_AcpTrak_0.Sector = &SectorTrackB;
					}

					MC_BR_RoutedMoveVel_AcpTrak_0.Velocity      = gTrakAsm.shuttle.parameter[gTrakAsm.status.shuttle_index].velocity;
					MC_BR_RoutedMoveVel_AcpTrak_0.RouteVelocity = gTrakAsm.shuttle.parameter[gTrakAsm.status.shuttle_index].velocity;
					MC_BR_RoutedMoveVel_AcpTrak_0.Acceleration  = gTrakAsm.shuttle.parameter[gTrakAsm.status.shuttle_index].accDec;
					MC_BR_RoutedMoveVel_AcpTrak_0.Deceleration  = gTrakAsm.shuttle.parameter[gTrakAsm.status.shuttle_index].accDec;
					MC_BR_RoutedMoveVel_AcpTrak_0.Jerk          = 0.0;
					MC_BR_RoutedMoveVel_AcpTrak_0.BufferMode    = mcABORTING;
					MC_BR_RoutedMoveVel_AcpTrak_0.AdvancedParameters.StartDirection     = mcDIR_UNDEFINED;
					MC_BR_RoutedMoveVel_AcpTrak_0.AdvancedParameters.EndDirection       = gTrakAsm.shuttle.parameter[gTrakAsm.status.shuttle_index].direction;
					MC_BR_RoutedMoveVel_AcpTrak_0.AdvancedParameters.ShuttleOrientation = mcDIR_UNDEFINED;

					gTrakAsm.actual_state = ACPt_CTRL_MOVE_VEL_2;
				}

				if(MC_BR_RoutedMoveVel_AcpTrak_0.Error == 1){
					MC_BR_AsmReset_AcpTrak_0.Execute = 1;
					gTrakAsm.actual_state = ACPt_CTRL_RESET_ERR;
				}
			}
			break;

		case ACPt_CTRL_MOVE_VEL_2: ///< Increase index by one (Velocity Control).
			{
				gTrakAsm.status.shuttle_index++;
				gTrakAsm.actual_state = ACPt_CTRL_MOVE_VEL_1;
			}
			break;

		case ACPt_CTRL_MOVE_POS_1: ///< Position control of the axes.
			{

				if(gTrakAsm.status.shuttle_index >= gTrakAsm.shuttle.num_of_shuttles){
					gTrakAsm.actual_state = ACPt_CTRL_WAIT;
				}else if(gTrakAsm.shuttle_axis[gTrakAsm.status.shuttle_index].controlif != 0){
					MC_BR_RoutedMoveAbs_AcpTrak_0.Axis          = &gTrakAsm.shuttle_axis[gTrakAsm.status.shuttle_index];
					MC_BR_RoutedMoveAbs_AcpTrak_0.Execute       = 1;

					if(gTrakAsm.shuttle.parameter[gTrakAsm.status.shuttle_index].sector_number == 0){
						MC_BR_RoutedMoveAbs_AcpTrak_0.Sector = &SectorTrackA;
					}else if(gTrakAsm.shuttle.parameter[gTrakAsm.status.shuttle_index].sector_number == 1){
						MC_BR_RoutedMoveAbs_AcpTrak_0.Sector = &SectorTrackB;
					}

					MC_BR_RoutedMoveAbs_AcpTrak_0.Position      = gTrakAsm.shuttle.parameter[gTrakAsm.status.shuttle_index].position;
					MC_BR_RoutedMoveAbs_AcpTrak_0.Velocity      = gTrakAsm.shuttle.parameter[gTrakAsm.status.shuttle_index].velocity;
					MC_BR_RoutedMoveAbs_AcpTrak_0.Acceleration  = gTrakAsm.shuttle.parameter[gTrakAsm.status.shuttle_index].accDec;
					MC_BR_RoutedMoveAbs_AcpTrak_0.Deceleration  = gTrakAsm.shuttle.parameter[gTrakAsm.status.shuttle_index].accDec;
					MC_BR_RoutedMoveAbs_AcpTrak_0.Jerk          = 0.0;
					MC_BR_RoutedMoveAbs_AcpTrak_0.BufferMode    = mcABORTING;
					MC_BR_RoutedMoveAbs_AcpTrak_0.AdvancedParameters.StartDirection     = mcDIR_UNDEFINED;
					MC_BR_RoutedMoveAbs_AcpTrak_0.AdvancedParameters.EndDirection       = gTrakAsm.shuttle.parameter[gTrakAsm.status.shuttle_index].direction;
					MC_BR_RoutedMoveAbs_AcpTrak_0.AdvancedParameters.ShuttleOrientation = mcDIR_UNDEFINED;

					gTrakAsm.actual_state = ACPt_CTRL_MOVE_POS_2;
				}

				if(MC_BR_RoutedMoveVel_AcpTrak_0.Error == 1){
					MC_BR_AsmReset_AcpTrak_0.Execute = 1;
					gTrakAsm.actual_state = ACPt_CTRL_RESET_ERR;
				}
			}
			break;

		case ACPt_CTRL_MOVE_POS_2: ///< Increase index by one (Position Control).
			{
				gTrakAsm.status.shuttle_index++;
				gTrakAsm.actual_state = ACPt_CTRL_MOVE_POS_1;
			}
			break;

		case ACPt_CTRL_STOPPING: ///< Stop each of the axes.
			{
				if(MC_Stop_0.Done == 1){
					gTrakAsm.status.shuttle_index++;
					MC_Stop_0.Execute = 0;
				}else if(gTrakAsm.shuttle_axis[gTrakAsm.status.shuttle_index].controlif != 0 && MC_Stop_0.Busy != 1){
					MC_Stop_0.Axis         = &gTrakAsm.shuttle_axis[gTrakAsm.status.shuttle_index];
					MC_Stop_0.Execute      = 1;
					MC_Stop_0.Deceleration = 20;
					MC_Stop_0.Jerk         = 0.0;
					MC_BR_RoutedMoveVel_AcpTrak_0.Execute = 0;
				}

				if(MC_Stop_0.Done == 1 && gTrakAsm.status.shuttle_index > gTrakAsm.shuttle.num_of_shuttles - 1){
					gTrakAsm.control.shuttle_stop = 0;
					gTrakAsm.actual_state = ACPt_CTRL_WAIT;
				}
			}
			break;

		case ACPt_CTRL_RESET_ERR: ///< The state machine is in an error state, wait for the automatic reset.
			{
				if(MC_BR_AsmReset_AcpTrak_0.Done == 1){
					gTrakAsm.control.shuttle_start = 0;
					gTrakAsm.control.shuttle_stop  = 0;
					MC_BR_AsmReset_AcpTrak_0.Execute      = 0;
					MC_BR_RoutedMoveVel_AcpTrak_0.Execute = 0;

					gTrakAsm.actual_state = ACPt_CTRL_WAIT;
				}
			}
			break;

		case ACPt_CTRL_DELETE: ///< Deleting each of the axes (shuttles) from the environment and returning to the initialization state.
			{
				MC_BR_AsmDeleteShuttle_AcpTrak_0.Command = mcACPTRAK_SH_DELETE_ALL;
				MC_BR_AsmDeleteShuttle_AcpTrak_0.Execute = 1;

				if(MC_BR_AsmDeleteShuttle_AcpTrak_0.Done == 1){
					gTrakAsm.actual_state = ACPt_CTRL_POWER_OFF;
				}
			}
			break;

	}

	/// set default parameters (change animation mode to default, null other parameters, etc.)
	if(gTrakAsm.control.default_shuttle_parameters == 1){
		gTrakAsm.control.animation_mode = ACPt_ANIM_MODE_1;
	}

	/// read output from the function block (the machine is active or not)
	gTrakAsm.status.active = MC_BR_AsmReadStatus_AcpTrak_0.AssemblyReady;

	/// read from mappview (HMI) -> set number of shuttles
	gTrakAsm.shuttle.num_of_shuttles = gTrakAsm.shuttle.num_of_shuttles_mv + 1;

	/**
	 * Digital-Twin camera control.
	 */

	if(dt_service.camera[0] == 1){
		/// Right Position
		dt_service.index = 0;
	}else if(dt_service.camera[1] == 1){
		/// Left Position
		dt_service.index = 1;
	}else if(dt_service.camera[2] == 1){
		/// Top Position
		dt_service.index = 2;
	}else if(dt_service.camera[3] == 1){
		/// Machine Vision 1 (Sector A)
		dt_service.index = 3;
	}else if(dt_service.camera[4] == 1){
		/// Machine Vision 2 (Sector B)
		dt_service.index = 4;
	}

	/**
	 * Call functions (FB) for control and data collection of each of the axes.
	 */

	/// This function block switches on the controllers for all segments of an assembly and identifies all shuttles.
	MC_BR_AsmPowerOn_AcpTrak(&MC_BR_AsmPowerOn_AcpTrak_0);
	MC_BR_AsmPowerOn_AcpTrak_0.Execute = 0;

	/// This function block switches off the controllers for all segments of an assembly.
	MC_BR_AsmPowerOff_AcpTrak(&MC_BR_AsmPowerOff_AcpTrak_0);

	/// This function block is used to create and add a shuttle to a defined position within a sector.
	/// This function is used if identification is not possible.
	MC_BR_SecAddShuttle_AcpTrak(&MC_BR_SecAddShuttle_AcpTrak_0);
	MC_BR_SecAddShuttle_AcpTrak_0.Execute = 0;

	/// This function block provides the axis reference of all shuttles in the assembly.
	MC_BR_AsmGetShuttle_AcpTrak(&MC_BR_AsmGetShuttle_AcpTrak_0);

	/// This function block can be used to start an elastic movement in the direction of a specified absolute position on a defined sector.
	/// This position is passed at the lower of the two velocity values at a maximum. The movement is performed continuously until the end of the target sector.
	MC_BR_RoutedMoveVel_AcpTrak(&MC_BR_RoutedMoveVel_AcpTrak_0);
	MC_BR_RoutedMoveVel_AcpTrak_0.Execute = 0;

	/// This function block can be used to start an elastic movement to a specified absolute position on a defined sector.
	MC_BR_RoutedMoveAbs_AcpTrak(&MC_BR_RoutedMoveAbs_AcpTrak_0);
	MC_BR_RoutedMoveAbs_AcpTrak_0.Execute = 0;

	/// This function block is used to determine the current state of the assembly.
	MC_BR_AsmReadStatus_AcpTrak(&MC_BR_AsmReadStatus_AcpTrak_0);
	MC_BR_AsmReset_AcpTrak(&MC_BR_AsmReset_AcpTrak_0);

	/// This function block deletes a shuttle and removes it from the assembly.
	MC_BR_AsmDeleteShuttle_AcpTrak(&MC_BR_AsmDeleteShuttle_AcpTrak_0);
	MC_BR_AsmDeleteShuttle_AcpTrak_0.Execute = 0;

	/// This function block performs a controlled movement stop and switches the axis to the Stopping state.
	MC_Stop(&MC_Stop_0);
}
```

#### Main.h - Init, cyclic, exit code
```c
/**
 * MIT License
 * Copyright(c) 2021 Roman Parak
 * Permission is hereby granted, free of charge, to any person obtaining a copy
 * of this software and associated documentation files (the "Software"), to deal
 * in the Software without restriction, including without limitation the rights
 * to use, copy, modify, merge, publish, distribute, sublicense, and/or sell
 * copies of the Software, and to permit persons to whom the Software is
 * furnished to do so, subject to the following conditions:
 * The above copyright notice and this permission notice shall be included in all
 * copies or substantial portions of the Software.
 * THE SOFTWARE IS PROVIDED "AS IS", WITHOUT WARRANTY OF ANY KIND, EXPRESS OR
 * IMPLIED, INCLUDING BUT NOT LIMITED TO THE WARRANTIES OF MERCHANTABILITY,
 * FITNESS FOR A PARTICULAR PURPOSE AND NONINFRINGEMENT. IN NO EVENT SHALL THE
 * AUTHORS OR COPYRIGHT HOLDERS BE LIABLE FOR ANY CLAIM, DAMAGES OR OTHER
 * LIABILITY, WHETHER IN AN ACTION OF CONTRACT, TORT OR OTHERWISE, ARISING FROM,
 * OUT OF OR IN CONNECTION WITH THE SOFTWARE OR THE USE OR OTHER DEALINGS IN THE
 * SOFTWARE.
 */

/**
 * Author   : Roman Parak
 * Email    : Roman.Parak@outlook.com
 * File Name: Main.h
 * Github   : https://github.com/rparak
 */

/** < Include B&R Automation libraries (declarations for B&R ANSI C extensions) */
#include <bur/plctypes.h>

/** < Include other libraries (mathematical functions, character string handling, etc.) */
#include <math.h>
#include <string.h>

#ifdef _DEFAULT_INCLUDES
#include <AsDefault.h>
#endif

/**
 * Main state machine for control of a ACOPOStrak.
 */
typedef enum acoposT_ctrl_state_enum{
	ACPt_CTRL_POWER_OFF, /**< Turn off the axes and reset each of the parameters. */
	ACPt_CTRL_POWER_ON, /**< Turn on each of the axes. */
	ACPt_CTRL_ADD_SHUTTLE_1, /**< Adding Shuttle for simulation. */
	ACPt_CTRL_ADD_SHUTTLE_2, /**< When the shuttle is added correctly, increase the index by one. */
	ACPt_CTRL_GET_SHUTTLE_1, /**< Get all available assembly information. (Initialization State) */
	ACPt_CTRL_GET_SHUTTLE_2, /**< Get all available assembly information. (Get next shuttle information) */
	ACPt_CTRL_GET_SHUTTLE_3, /**< Get all available assembly information. (When the shuttle is exist, increase the index by one) */
	ACPt_CTRL_WAIT, /**< Wait for command from HMI visualization (user). */
	ACPt_CTRL_MOVE_VEL_1, /**< Velocity control of the axes. */
	ACPt_CTRL_MOVE_VEL_2, /**< Increase index by one (Velocity Control). */
	ACPt_CTRL_MOVE_POS_1, /**< Position control of the axes. */
	ACPt_CTRL_MOVE_POS_2, /**< Increase index by one (Position Control). */
	ACPt_CTRL_STOPPING, /**< Stop each of the axes. */
	ACPt_CTRL_RESET_ERR, /**< The state machine is in an error state, wait for the automatic reset. */
	ACPt_CTRL_DELETE /**< Deleting each of the axes (shuttles) from the environment and returning to the initialization state. */
}acoposT_ctrl_state_enum;

/**
 * Main state machine for animation mode control of a ACOPOStrak.
 */
typedef enum acoposT_animMode_state_enum{
	ACPt_ANIM_MODE_1, /**< Animation Mode 1 - Velocity control (around the specified sector). */
	ACPt_ANIM_MODE_2, /**< Animation Mode 2 - Position control (around the Sector A, stop under the machine vision camera). */
	ACPt_ANIM_MODE_3, /**< Animation Mode 3 - Position control (around the Sector B, stop under the machine vision camera). */
	ACPt_ANIM_MODE_4 /**< Animation Mode 4 - Velocity control (around both sectors). */
}acoposT_animMode_state_enum;

/**
 * Command execution structure for control of a machine ACOPOStrak.
 */
typedef struct TrakAsm_ctrl_command{
	BOOL power; /**< Power on. */
	BOOL reset_evn; /**< Reset environment. */
	BOOL shuttle_start; /**< Start movement. */
	BOOL shuttle_stop; /**< Stop movement. */
	BOOL default_shuttle_parameters; /**< Set default parameters. */
	acoposT_animMode_state_enum animation_mode; /**< Animation Mode - Enum. */
	acoposT_animMode_state_enum animation_mode_before; /**< Animation Mode - Enum. */
}TrakAsm_ctrl_command;

/**
 * Main state machine for animation mode control of a ACOPOStrak.
 */
typedef struct TrakAsm_parameter_shuttle{
	LREAL initial_position; /**< Initial Position of the shuttle. */
	USINT sector_number; /**< Sector Number: 0 - Sector A, 1 - Sector  */
	USINT direction; /**< Movement direction: 0 - Positive, 1 - Negative */
	LREAL position; /**< Target position. */
	REAL velocity; /**< Target velocity. */
	REAL accDec; /**< Target acceleration/deceleration -> same value. */
}TrakAsm_parameter_shuttle;

/**
 * Structure for shuttle parameters.
 */
typedef struct TrakAsm_shuttle{
	USINT num_of_shuttles; /**< Number of shuttles. */
	USINT num_of_shuttles_mv; /**< Number of shuttles (from mappview). */
	REAL shuttle_offset; /**< Initial shuttle offset. */
	LREAL sector_legth; /**< Sector length - in our experiment, both have the same value. */
	USINT move_type; /**< Move type: 0 - Move Velocity, 1 - Move Position */
	USINT initial_sector; /**< Initial sector of the start of the movement. */
	REAL shuttle_velocity; /**< Target velocity of the shuttle. */
	TrakAsm_parameter_shuttle parameter[6];
}TrakAsm_shuttle;

/**
 * Structure for ACOPOStrak status information.
 */
typedef struct TrakAsm_status_command{
	BOOL power_on; /**< The machine is power on. */
	BOOL active;  /**< The machine is active. */
	BOOL is_homed; /**< The shuttles of the machine are homed. */
	BOOL shuttles_exist; /**< There are one or more shuttles. */
	USINT shuttle_index; /**< Controlled shuttle index. */
}TrakAsm_status_command;

/**
 * Structure for shuttle data collection.
 */
typedef struct TrakAsm_data_collection{
	LREAL position; /**< Current position. */
	REAL velocity; /**< Current velocity. */
	USINT sector; /**< Current sector. */
	USINT number_of_rotates; /**< Number of rotates (around the sector). */
}TrakAsm_data_collection;

/**
 * Custom structure for digital-twin service (camera control, machine vision position, etc.)
 */
typedef struct DigitalTwin_service{
	BOOL camera[5]; /**< Camera control (index): 0 - right, 1 - left, 2 - up, 3 - machine vision (Sector A), 4 - machine vision (Sector B) */
	USINT index; /**< Index for Digital-Twin. */
	LREAL machine_vision_position[2]; /**< Initial position under the machine vision camera in the current sector: 0 - Sector A, 1 - Sector B */
}DigitalTwin_service;

/**
 * Custom structure for controlling some MappView functions.
 */
typedef struct mappView_service{
	BOOL enable_param; /**< Enable/disable of widgets. */
}mappView_service;

/**
 * Custom structure for ACOPOStrak control and data collection.
 */
typedef struct TrakAsm_ctrl_main{
	TrakAsm_ctrl_command control;
	TrakAsm_shuttle shuttle;
	TrakAsm_status_command status;
	TrakAsm_data_collection data_collection[6];
	McAxisType shuttle_axis[6];
	acoposT_ctrl_state_enum actual_state;
}TrakAsm_ctrl_main;

/**
* Function blocks for smooth control of the ACOPOStrak machine (for more information, see Help 'F1').
*/
_LOCAL struct MC_BR_AsmPowerOn_AcpTrak MC_BR_AsmPowerOn_AcpTrak_0;
_LOCAL struct MC_BR_AsmPowerOff_AcpTrak MC_BR_AsmPowerOff_AcpTrak_0;
_LOCAL struct MC_BR_SecAddShuttle_AcpTrak MC_BR_SecAddShuttle_AcpTrak_0;
_LOCAL struct MC_BR_AsmGetShuttle_AcpTrak MC_BR_AsmGetShuttle_AcpTrak_0;
_LOCAL struct MC_BR_RoutedMoveVel_AcpTrak MC_BR_RoutedMoveVel_AcpTrak_0;
_LOCAL struct MC_BR_RoutedMoveAbs_AcpTrak MC_BR_RoutedMoveAbs_AcpTrak_0;
_LOCAL struct MC_BR_AsmDeleteShuttle_AcpTrak MC_BR_AsmDeleteShuttle_AcpTrak_0;
_LOCAL struct MC_BR_AsmReadStatus_AcpTrak MC_BR_AsmReadStatus_AcpTrak_0;
_LOCAL struct MC_BR_AsmReset_AcpTrak MC_BR_AsmReset_AcpTrak_0;
_LOCAL struct MC_Stop MC_Stop_0;
_LOCAL struct MC_BR_ShReadInfo_AcpTrak MC_BR_ShReadInfo_AcpTrak_ID[6];
_LOCAL struct MC_BR_ShReadInfo_AcpTrak MC_BR_ShReadInfo_AcpTrak_NULL;

/// Custom structure for digital-twin service (camera control, machine vision position, etc.)
_LOCAL DigitalTwin_service dt_service;
/// Custom structure for ACOPOStrak control and data collection.
_LOCAL TrakAsm_ctrl_main gTrakAsm;
/// Custom structure for controlling some MappView functions (enable/disable of widgets, etc.)
_LOCAL mappView_service mv_service;

/// auxiliary counter (animation mode 2 - 3)
_LOCAL USINT animation_aux_counter;

void reset_shuttle_param(USINT num_of_shuttles, USINT initial_sector, REAL offset){
	/**
	Description:
		Function to reset each of the parameters.

	Args:
		(1) num_of_shuttles [USINT]: Number of the shuttles.
		(2) initial_sector [USINT]: Initial sector of the start of the movement.
		(3) offset [REAL]: Initial shuttle offset.
	*/

	int i;

	for(i = 0; i < (int)(sizeof(gTrakAsm.shuttle.parameter)/sizeof(gTrakAsm.shuttle.parameter[0])); i++){
		if(i < num_of_shuttles){
			gTrakAsm.shuttle.parameter[i].initial_position = (i + 1) * offset;
			gTrakAsm.shuttle.parameter[i].sector_number = initial_sector;

			if(initial_sector == 0){
				gTrakAsm.shuttle.parameter[i].direction     = 0;
			}else if(initial_sector == 1){
				gTrakAsm.shuttle.parameter[i].direction     = 1;
			}
			gTrakAsm.shuttle.parameter[i].position      = 1.0;
			gTrakAsm.shuttle.parameter[i].velocity      = gTrakAsm.shuttle.shuttle_velocity;
			gTrakAsm.shuttle.parameter[i].accDec  		= gTrakAsm.shuttle.shuttle_velocity*10;
		}else{
			gTrakAsm.shuttle.parameter[i].initial_position = 0.0;
			gTrakAsm.shuttle.parameter[i].sector_number = 0;
			gTrakAsm.shuttle.parameter[i].direction     = 0;
			gTrakAsm.shuttle.parameter[i].position      = 0.0;
			gTrakAsm.shuttle.parameter[i].velocity      = 0.0;
			gTrakAsm.shuttle.parameter[i].accDec  		= 0.0;
		}
	}

	gTrakAsm.control.animation_mode = ACPt_ANIM_MODE_1;
}

void reset_env(){
	/**
	Description:
		Function to reset environment (clear the shuttles from the Digital-Twin).
	*/

	int i;

	for(i = 0; i < (int)(sizeof(gTrakAsm.data_collection)/sizeof(gTrakAsm.data_collection[0])); i++){
		gTrakAsm.data_collection[i].position = 0.0;
		gTrakAsm.data_collection[i].velocity = 0.0;
		gTrakAsm.data_collection[i].number_of_rotates = 0;
		/// Global Variable Reset
		gShuttleMon.Shuttle[i].Position.X 	      = 0.0;
		gShuttleMon.Shuttle[i].Position.Y 		  = 0.0;
		gShuttleMon.Shuttle[i].Orientation.Angle1 = 0.0;
		/// Reset the data collection function block
		MC_BR_ShReadInfo_AcpTrak_ID[i] = MC_BR_ShReadInfo_AcpTrak_NULL;
	}
}

void read_shuttle_param(USINT num_of_shuttles, REAL offset){
	/**
	Description:
		Function for reading shuttle parameters (position, velocity, etc.) and calculating the absolute position, number of rotation, etc., of the current sector.

	Args:
		(1) num_of_shuttles [USINT]: Number of the shuttles.
		(2) offset [REAL]: Initial shuttle offset.
	*/

	int i;

	for(i = 0; i < (int)(sizeof(gTrakAsm.shuttle.parameter)/sizeof(gTrakAsm.shuttle.parameter[0])); i++){
		if(i < num_of_shuttles){
			MC_BR_ShReadInfo_AcpTrak_ID[i].Enable = 1;
			MC_BR_ShReadInfo_AcpTrak_ID[i].Axis   = &gTrakAsm.shuttle_axis[i];
			/// Call Function Block
			MC_BR_ShReadInfo_AcpTrak(&MC_BR_ShReadInfo_AcpTrak_ID[i]);

			if(fabs(MC_BR_ShReadInfo_AcpTrak_ID[i].ShuttleInfo.CurrentValues.Position) <= gTrakAsm.shuttle.sector_legth){
				gTrakAsm.data_collection[i].number_of_rotates = 0;
				gTrakAsm.data_collection[i].position          = fabs(MC_BR_ShReadInfo_AcpTrak_ID[i].ShuttleInfo.CurrentValues.Position);
			}else{
				gTrakAsm.data_collection[i].number_of_rotates = (USINT)floor(((MC_BR_ShReadInfo_AcpTrak_ID[i].ShuttleInfo.LifeCycleInfo.AbsoluteMovementDistance + ((i + 1) * offset)) / gTrakAsm.shuttle.sector_legth));
				gTrakAsm.data_collection[i].position 	      = ((MC_BR_ShReadInfo_AcpTrak_ID[i].ShuttleInfo.LifeCycleInfo.AbsoluteMovementDistance + ((i + 1) * offset)) - (gTrakAsm.shuttle.sector_legth * (gTrakAsm.data_collection[i].number_of_rotates)));
			}

			gTrakAsm.data_collection[i].velocity = MC_BR_ShReadInfo_AcpTrak_ID[i].ShuttleInfo.CurrentValues.Velocity;

			if(strcmp(MC_BR_ShReadInfo_AcpTrak_ID[i].ShuttleInfo.CurrentValues.SectorName, "SectorTrackA") == 0){
				gTrakAsm.data_collection[i].sector = 0;
			}else if(strcmp(MC_BR_ShReadInfo_AcpTrak_ID[i].ShuttleInfo.CurrentValues.SectorName, "SectorTrackB") == 0){
				gTrakAsm.data_collection[i].sector = 1;
			}else{
				gTrakAsm.data_collection[i].sector = 10;
			}
		}
	}
}

void set_shuttle_move_param(USINT index, USINT sector, LREAL position, REAL velocity){
	/**
	Description:
		Function for setting the parameters of the shuttle's movement.

	Args:
		(1) index [USINT]: Index of the current shuttle.
		(1) sector [USINT]: Movement in the sector (0 - Sector A, 1 - Sector B).
		(1) position [LREAL]: Target position of the shuttle.
		(1) velocity [REAL]: Target velocity of the shuttle.
	*/

	gTrakAsm.shuttle.parameter[index].sector_number = sector;

	if(sector == 0){
		gTrakAsm.shuttle.parameter[index].direction     = 0;
	}else if(sector == 1){
		gTrakAsm.shuttle.parameter[index].direction     = 1;
	}

	gTrakAsm.shuttle.parameter[index].position      = position;
	gTrakAsm.shuttle.parameter[index].velocity      = velocity;
	gTrakAsm.shuttle.parameter[index].accDec  		= velocity*10;
}

USINT min_number_index(USINT num_of_shuttles, LREAL machine_vision_position, USINT sector){
	/**
	Description:
		Auxiliary function for calculating the minimum position index of the shuttle.

	Args:
		(1) num_of_shuttles [USINT]: Number of the shuttles.
		(2) machine_vision_position [LREAL]: Position of the machine vision camer in the digital-twin.
		(3) sector [USINT]: Sector number for calculation (0 - Sector A, 1 - Sector B).

	Returns:
		(1) parameter{1} [USINT]: Resulting index (0 .. num_of_shuttles - 1, 100 -> error).
	*/

	LREAL min_num = 10.0;
	USINT index = 100;

	int i = 0;

	for(i = 0; i < (int)(sizeof(gTrakAsm.data_collection)/sizeof(gTrakAsm.data_collection[0])); i++){
		if(i < num_of_shuttles){
			if(gTrakAsm.data_collection[i].position <= min_num && gTrakAsm.data_collection[i].position != machine_vision_position && gTrakAsm.data_collection[i].sector == sector){
				min_num = gTrakAsm.data_collection[i].position;
				index   = i;
			}
		}
	}

	return index;
}

USINT max_number_index(USINT num_of_shuttles, LREAL machine_vision_position, USINT sector){
	/**
	Description:
		Auxiliary function for calculating the maximum position index of the shuttle.

	Args:
		(1) num_of_shuttles [USINT]: Number of the shuttles.
		(2) machine_vision_position [LREAL]: Position of the machine vision camer in the digital-twin.
		(3) sector [USINT]: Sector number for calculation (1 - Sector A, 2 - Sector B).

	Returns:
		(1) parameter{1} [USINT]: Resulting index (0 .. num_of_shuttles - 1, 100 -> error).
	*/

	LREAL max_num = -1.0;
	USINT index   = 100;

	int i = 0;

	for(i = 0; i < (int)(sizeof(gTrakAsm.data_collection)/sizeof(gTrakAsm.data_collection[0])); i++){
		if(i < num_of_shuttles){
			if(gTrakAsm.data_collection[i].position >= max_num && gTrakAsm.data_collection[i].position != machine_vision_position && gTrakAsm.data_collection[i].sector == sector){
				max_num = gTrakAsm.data_collection[i].position;
				index   = i;
			}
		}
	}

	return index;
}

void set_animation_mode(){

	/**
	 * Main state machine for animation mode control of a ACOPOStrak.
	 *
	 * Number of states: 4
	 * Structure: acoposT_animMode_state_enum
	 *
	 * Note:
	 * Sector B has the initial opposite direction as in sector A, so the first shuttle is the minimum index.
	 * In sector A, this is the maximum index.
	 */

	switch(gTrakAsm.control.animation_mode){
		case ACPt_ANIM_MODE_1: /**< Animation Mode 1 - Velocity control (around the specified sector). */
			{
				gTrakAsm.control.animation_mode_before = ACPt_ANIM_MODE_1;
				/// Type (0) -> Move Velocity
				gTrakAsm.shuttle.move_type             = 0;

				if(gTrakAsm.control.shuttle_start == 1){
					reset_shuttle_param(gTrakAsm.shuttle.num_of_shuttles, gTrakAsm.shuttle.initial_sector, gTrakAsm.shuttle.shuttle_offset);
				}
			}
			break;

		case ACPt_ANIM_MODE_2: /**< Animation Mode 2 - Position control (around the Sector A, stop under the machine vision camera). */
			{
				if(gTrakAsm.control.animation_mode != gTrakAsm.control.animation_mode_before){
					animation_aux_counter = 0;
					gTrakAsm.control.animation_mode_before = ACPt_ANIM_MODE_2;
				}

				/// Type (1) -> Move Position
				gTrakAsm.shuttle.move_type = 1;

				if(gTrakAsm.control.shuttle_start == 1){
					/// find the first shuttle from the train (the first scan in sector A because the final position of the shuttles is in sector A)
					animation_aux_counter = max_number_index(gTrakAsm.shuttle.num_of_shuttles, dt_service.machine_vision_position[0], 0);

					if(animation_aux_counter == 100){
						/// the second scan is in sector B
						animation_aux_counter = min_number_index(gTrakAsm.shuttle.num_of_shuttles, dt_service.machine_vision_position[1], 1);
					}

					int i;

					for(i = 0; i < (int)(sizeof(gTrakAsm.shuttle.parameter)/sizeof(gTrakAsm.shuttle.parameter[0])); i++){
						if(i < gTrakAsm.shuttle.num_of_shuttles){
							if(i == animation_aux_counter){
								/// stop under the machine vision camera (the variable *.machine_vision_position[0] is initialized in 'Main.c')
								set_shuttle_move_param(i, 0, dt_service.machine_vision_position[0], gTrakAsm.shuttle.shuttle_velocity);
							}else{
								/// stop one meter in front of the machine vision camera (the last shuttle position is *.machine_vision_position[0] - 1, other positions are calculated automatically from FB without collision)
								set_shuttle_move_param(i, 0, dt_service.machine_vision_position[1] - 1.0, gTrakAsm.shuttle.shuttle_velocity);
							}
						}
					}
				}
			}
			break;

		case ACPt_ANIM_MODE_3: /**< Animation Mode 3 - Position control (around the Sector B, stop under the machine vision camera). */
			{
				if(gTrakAsm.control.animation_mode != gTrakAsm.control.animation_mode_before){
					animation_aux_counter = 0;
					gTrakAsm.control.animation_mode_before = ACPt_ANIM_MODE_3;
				}

				/// Type (1) -> Move Position
				gTrakAsm.shuttle.move_type = 1;

				if(gTrakAsm.control.shuttle_start == 1){
					/// find the first shuttle from the train (the first scan in sector B because the final position of the shuttles is in sector B)
					animation_aux_counter = min_number_index(gTrakAsm.shuttle.num_of_shuttles, dt_service.machine_vision_position[1], 1);

					if(animation_aux_counter == 100){
						/// the second scan is in sector A
						animation_aux_counter = max_number_index(gTrakAsm.shuttle.num_of_shuttles, dt_service.machine_vision_position[0], 0);
					}

					int i;

					for(i = 0; i < (int)(sizeof(gTrakAsm.shuttle.parameter)/sizeof(gTrakAsm.shuttle.parameter[0])); i++){
						if(i < gTrakAsm.shuttle.num_of_shuttles){
							if(i == animation_aux_counter){
								/// stop under the machine vision camera (the variable *.machine_vision_position[1] is initialized in 'Main.c')
								set_shuttle_move_param(i, 1, dt_service.machine_vision_position[1], gTrakAsm.shuttle.shuttle_velocity);
							}else{
								/// stop one meter in front of the machine vision camera (the last shuttle position is *.machine_vision_position[1] - 1, other positions are calculated automatically from FB without collision)
								set_shuttle_move_param(i, 1, dt_service.machine_vision_position[1] + 1.0, gTrakAsm.shuttle.shuttle_velocity);
							}
						}
					}
				}
			}
			break;

		case ACPt_ANIM_MODE_4: /**< Animation Mode 4 - Velocity control (around both sectors). */
			{
				gTrakAsm.control.animation_mode_before = ACPt_ANIM_MODE_4;
				/// Type (0) -> Move Velocity
				gTrakAsm.shuttle.move_type = 0;

				int i;

				if(gTrakAsm.control.shuttle_start == 1){
					for(i = 0; i < (int)(sizeof(gTrakAsm.shuttle.parameter)/sizeof(gTrakAsm.shuttle.parameter[0])); i++){
						/// division of shuttles between individual sectors
						if(i < gTrakAsm.shuttle.num_of_shuttles){
							if(i % 2 == 0){
								set_shuttle_move_param(i, 0, 1.0, gTrakAsm.shuttle.shuttle_velocity);
							}else{
								set_shuttle_move_param(i, 1, 1.0, gTrakAsm.shuttle.shuttle_velocity);
							}
						}
					}
				}
			}
			break;

	}
}
```

- Visualisation Logical/mappView (not shown)

Listed in the project but not available here: Logical/Global.typ, Logical/Technology/tCTRL_m/Types.typ, Logical/Technology/tCTRL_m/Variables.var
